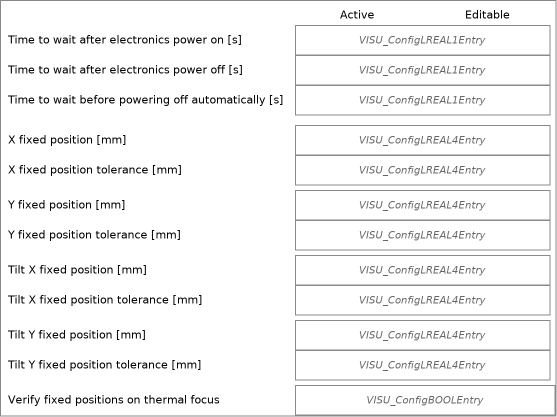
VISUALIZATION VISU_M2Config_General  // 557x417
VAR_IN_OUT
    editable : M2Config;
	active : M2Config;
END_VAR
    Label (295,5 125x20), "Active"
    Label (425,5 125x20), "Editable"
    Label (5,25 250x30), "Time to wait after electronics power on [s]"
    Frame (295,25 255x30)
        shows VISU_ConfigLREAL1Entry(active := active.waitAfterPowerOn, editable := editable.waitAfterPowerOn)
    Label (5,55 250x30), "Time to wait after electronics power off [s]"
    Frame (295,55 255x30)
        shows VISU_ConfigLREAL1Entry(active := active.waitAfterPowerOff, editable := editable.waitAfterPowerOff)
    Label (5,85 285x30), "Time to wait before powering off automatically [s]"
    Frame (295,85 255x30)
        shows VISU_ConfigLREAL1Entry(active := active.powerOffTimeout, editable := editable.powerOffTimeout)
    Frame (295,125 255x30)
        shows VISU_ConfigLREAL4Entry(active := active.fixedXPosition, editable := editable.fixedXPosition)
    Label (5,125 285x30), "X fixed position [mm]"
    Label (5,155 285x30), "X fixed position tolerance [mm]"
    Frame (295,155 255x30)
        shows VISU_ConfigLREAL4Entry(active := active.fixedXPositionTolerance, editable := editable.fixedXPositionTolerance)
    Frame (295,190 255x30)
        shows VISU_ConfigLREAL4Entry(active := active.fixedYPosition, editable := editable.fixedYPosition)
    Label (5,190 285x30), "Y fixed position [mm]"
    Label (5,220 285x30), "Y fixed position tolerance [mm]"
    Frame (295,220 255x30)
        shows VISU_ConfigLREAL4Entry(active := active.fixedYPositionTolerance, editable := editable.fixedYPositionTolerance)
    Frame (295,255 255x30)
        shows VISU_ConfigLREAL4Entry(active := active.fixedTiltXPosition, editable := editable.fixedTiltXPosition)
    Label (5,255 285x30), "Tilt X fixed position [mm]"
    Label (5,285 285x30), "Tilt X fixed position tolerance [mm]"
    Frame (295,285 255x30)
        shows VISU_ConfigLREAL4Entry(active := active.fixedTiltXPositionTolerance, editable := editable.fixedTiltXPositionTolerance)
    Frame (295,320 255x30)
        shows VISU_ConfigLREAL4Entry(active := active.fixedTiltYPosition, editable := editable.fixedTiltYPosition)
    Label (5,320 285x30), "Tilt Y fixed position [mm]"
    Label (5,350 285x30), "Tilt Y fixed position tolerance [mm]"
    Frame (295,350 255x30)
        shows VISU_ConfigLREAL4Entry(active := active.fixedTiltYPositionTolerance, editable := editable.fixedTiltYPositionTolerance)
    Label (5,385 285x30), "Verify fixed positions on thermal focus"
    Frame (295,385 260x30)
        shows VISU_ConfigBOOLEntry(active := active.verifyFixedPositinsOnThermalFocus, editable := editable.verifyFixedPositinsOnThermalFocus)
END_VISUALIZATION

(* stored: Version 1.1.0.1, ProductVersion 3.1.4019.2
   Visu VISU_M2Config_General: Id {c2e9f574-c79f-49ff-898d-e65d387ff985} *)
